TYPE STATUS :
STRUCT
	MoveActive			:BOOL;
	eStop				:BOOL;
	
	Rack_Err			:BOOL	:= FALSE;
	Script_Open_Err		:BOOL	:= FALSE;	
	Script_Read_Err		:BOOL	:= FALSE;
	List_Overflow_Err	:BOOL	:= FALSE;
	Move_Rel_Err		:BOOL 	:= FALSE;
	Move_Abs_Err		:BOOL	:= FALSE;
	//HS_Err				:BOOL	:= FALSE;
	Basin_Exceed_Err	:BOOL	:= FALSE;
	//Basin_Set_Err		:BOOL	:= FALSE;
	
	
	AxesLocated			:BOOL	:= FALSE;
	//HardStopLoc			:BOOL	:= FALSE; 
	//zSafeSet			:BOOL	:= FALSE;
	//BasinSet			:BOOL	:= FALSE;
	Stop_Int			:BOOL	:= FALSE;
	PowerError			:BOOL	:= FALSE;
	
	CurInstr			:INT;
	NextInstr			:INT;
	ScriptEnd			:INT;
	RUN_INDEX			:INT;
	
	xCoupled			:BOOL;
	xPosOut				:LREAL;
	xVelOut				:LREAL;
	yPosOut				:LREAL;
	yVelOut				:LREAL;
	zPosOut				:LREAL;
	zVelOut				:LREAL;
	
	basinxMin			:LREAL;
	basinxMax			:LREAL;
	basinyMin			:LREAL;
	basinyMax			:LREAL;
	basinstate			:INT	:= 0;

	
	HardStopLocations	:ARRAY[0..2] OF LREAL	:= [100000,8991,1000]; //includes carriage offsets 
	CARRIAGE_OFFSETS	:ARRAY[0..2] OF LREAL	:= [500,250,100]; //for display. also in GVL_MOTION
	
	
END_STRUCT
END_TYPE

(* stored: Version 1.1.0.1, ProductVersion 3.1.4026.18
   DUT STATUS: Id {f85b29e1-bc75-46b4-af59-e2e0fcb03fd0} *)
